(* Logix 5000 project; controller SIM_IO Emulate 5570 rev 30.12; software revision 30.01 *)

TASK MainTask (continuous, watchdog 500 ms) : MainProgram

MODULES
   Local : Emulate 5570 (ICP 2, rev 30.12)
      SIM : vendor 1 type 0 code 15 (ICP 3, rev 1.1, Output RPI 50 ms)
END_MODULES

PROGRAM MainProgram   (* main routine MainRoutine *)
VAR
   Motor : ALIAS FOR Local:3:O.Data[0].0;
   Start : ALIAS FOR Local:3:I.Data[1].0;
   Stop : ALIAS FOR Local:3:I.Data[1].1;
END_VAR

ROUTINE MainRoutine   (* ladder *)
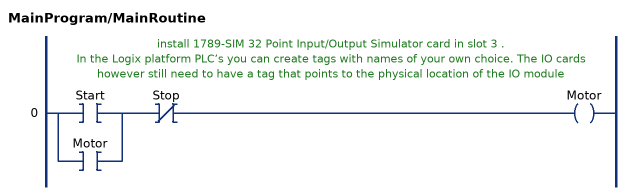
   // install 1789-SIM 32 Point Input/Output Simulator card in slot 3 .
   // In the Logix platform PLC’s you can create tags with names of your own choice. The IO cards however still need to have a tag that points to the physical location of the IO module
   0: [XIC(Start) ,XIC(Motor) ]XIO(Stop)OTE(Motor);
END_ROUTINE
END_PROGRAM
